{attribute 'qualified_only'}
VAR_GLOBAL
	// xDO%115.0_A5_5
	SST_MV_weiss AT %Q*: BOOL;
	// xDO%115.1_A5_5
	SST_MV_rot AT %Q*: BOOL;
	// xDO%115.2_A5_5
	SST_MV_blau AT %Q*: BOOL;
	// iAI%130.0_A5_4
	SST_Farbsensor AT %I*: INT;
	// xDI%138.4_A5_1
	SST_Impulstaster AT %I*: BOOL;
	// xDI%138.5_A5_1
	SST_LS_Eingang AT %I*: BOOL;
	// xDI%138.6_A5_1
	SST_LS_nach_Farbsensor AT %I*: BOOL;
	// xDI%138.7_A5_1
	SST_LS_weiss AT %I*: BOOL;
	// xDI%139.0_A5_1
	SST_LS_rot AT %I*: BOOL;
	// xDI%139.1_A5_1
	SST_LS_blau AT %I*: BOOL;
	// xDO%114.6_A5_2
	SST_MOT_Foerderband AT %Q*: BOOL;
	// xDO%114.7_A5_8
	SST_Kompressor AT %Q*: BOOL;
END_VAR

(* stored: Version 1.1.0.1, ProductVersion 3.1.4024.15
   GVL GVL_SST: Id {e2d210c6-cb47-4b21-a087-975f3e114acc} *)
